TEXTLIST TL_E_MOVER_SELECTOR
  0 = 'SELECT_MOVER_INDEX'
  1 = 'SELECT_MOVER_AXIS_ID'
   = ''
END_TEXTLIST

(* stored: Version 1.1.0.1, ProductVersion 3.1.4026.13
   TextList TL_E_MOVER_SELECTOR: Id {7a3072b9-4251-46df-8d96-80d87408c858} *)
